FUNCTION_BLOCK FB_Kommunikation
VAR_INPUT
	I_sIP		:STRING;
	SW			:SystemStatusWord;
END_VAR

VAR_OUTPUT
	CW			:SystemControlWord;
	Busy		:BOOL;
	Error		:BOOL;
	ErrorID		:DWORD;
END_VAR

VAR
	Connect				:UA_Connect;
	Disconnect			:UA_Disconnect; 
	Read 				:UA_Read;
	Write				:UA_Write;
	Node				:UA_NodeGetHandle;
	NameSpaceIndex		:UA_GetNamespaceIndex;
	
	ConnectInfo			:ST_UASessionConnectInfo;
	NodeID				:ST_UANodeID;
	NodeInfo			:ST_UANodeAdditionalInfo;
	
	ConnectionHdl		:DWORD;
	NoteHdl				:DWORD;
	NameSpace			:UINT;
	IndexRangeCount		:UINT := 1;
	IndexRange			:ARRAY [1..nMaxIndexRange] OF ST_UAIndexRange;
	NodeIdentifier		:STRING(MAX_STRING_LENGTH) := 'GVL_OPC_UA.SW';
	ReadData			:SystemStatusWord; 		// change to node data type
END_VAR

// Definition der Verbindungsinformationen
ConnectInfo.tSessionTimeout := T#1M;
ConnectInfo.tConnectTimeout := T#1M;
ConnectInfo.sApplicationName := '';
ConnectInfo.eSecurityMode := eUASecurityMsgMode_Sign_Encrypt;				// 3 = Sign_Encrypted
ConnectInfo.eSecurityPolicyUri := eUASecurityPolicy_Basic256Sha256;			// 4 = Basic256  
ConnectInfo.eTransportProfileUri := eUATransportProfileUri_UATcp;			// 1 = UATcp
ConnectInfo.stUserIdentTokenType.eUserIdentTokenType := eUAUITT_Username;	// 1 = Username
ConnectInfo.stUserIdentTokenType.sTokenParam1 := 'Administrator';			// Username
ConnectInfo.stUserIdentTokenType.sTokenParam2 := '1';						// PW

GVL.SW := ReadData;

ACTION ACT_Connect:
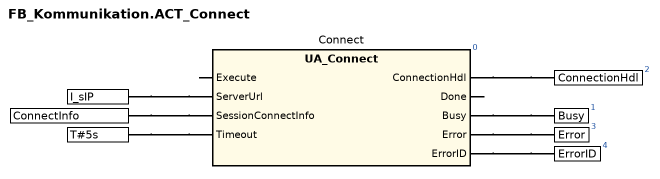
Connect(ServerUrl := I_sIP, SessionConnectInfo := ConnectInfo, Timeout := T#5s); // UA_Connect
Busy := Connect.Busy;
ConnectionHdl := Connect.ConnectionHdl;
Error := Connect.Error;
ErrorID := Connect.ErrorID;
END_ACTION

ACTION ACT_Disconnect:
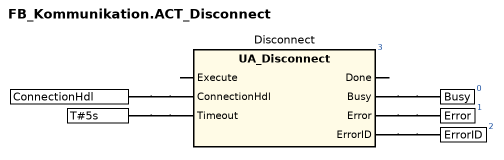
Busy := Disconnect.Busy;
Error := Disconnect.Error;
ErrorID := Disconnect.ErrorID;
Disconnect(ConnectionHdl := ConnectionHdl, Timeout := T#5s); // UA_Disconnect
END_ACTION

ACTION ACT_GetNameSpaceIndex:
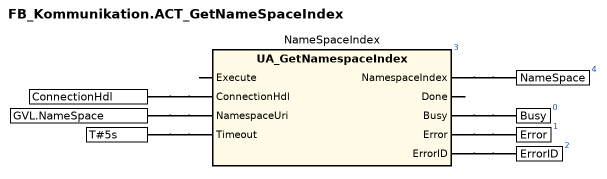
Busy := NameSpaceIndex.Busy;
Error := NameSpaceIndex.Error;
ErrorID := NameSpaceIndex.ErrorID;
NameSpaceIndex(ConnectionHdl := ConnectionHdl, NamespaceUri := GVL.NameSpace, Timeout := T#5s); // UA_GetNamespaceIndex
NameSpace := NameSpaceIndex.NamespaceIndex;
END_ACTION

ACTION ACT_GetNodes:
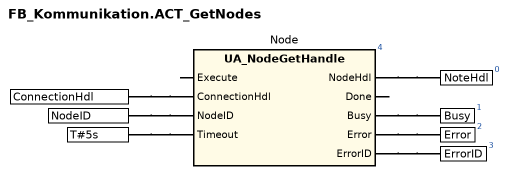
NoteHdl := Node.NodeHdl;
Busy := Node.Busy;
Error := Node.Error;
ErrorID := Node.ErrorID;
Node(ConnectionHdl := ConnectionHdl, NodeID := NodeID, Timeout := T#5s); // UA_NodeGetHandle
END_ACTION

ACTION ACT_Read:
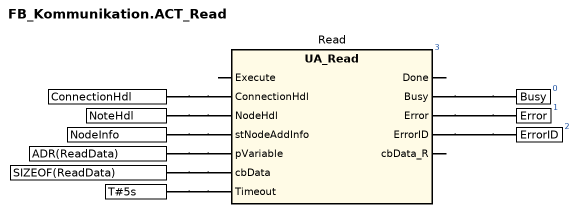
Busy := Read.Busy;
Error := Read.Error;
ErrorID := Read.ErrorID;
Read(
    ConnectionHdl := ConnectionHdl,
    NodeHdl := NoteHdl,
    stNodeAddInfo := NodeInfo,
    pVariable := ADR(ReadData),
    cbData := SIZEOF(ReadData),
    Timeout := T#5s); // UA_Read
END_ACTION

ACTION ACT_Write:
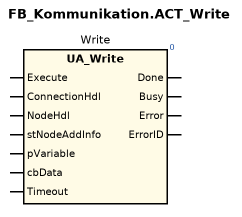
Write(); // UA_Write
END_ACTION

METHOD M_M_Connect : BOOL
VAR_INPUT
END_VAR
// Setzen der Ausführvariabel
Connect.Execute := TRUE;
// Aufrufen der Aktion
ACT_Connect();

// Methode abschliessen
IF Connect.Done THEN
	Connect.Execute := FALSE;
	M_M_Connect := TRUE;
END_IF
END_METHOD

METHOD M_M_Disconnect : BOOL
VAR_INPUT
END_VAR
// Setzen der Ausführvariabel
Disconnect.Execute := TRUE;
// Aufrufen der Aktion
Act_Disconnect();

// Methode abschliessen
IF Disconnect.Done THEN
	Disconnect.Execute := FALSE;
	M_M_Disconnect := TRUE;
END_IF
END_METHOD

METHOD M_M_GetNameSpaceIndex : BOOL
VAR_INPUT
END_VAR
// Setzen der Ausführvariabel
NameSpaceIndex.Execute := TRUE;
// Aufrufen der Aktion
ACT_GetNameSpaceIndex();

// Methode abschliessen
IF NameSpaceIndex.Done THEN
	NameSpaceIndex.Execute := FALSE;
	M_M_GetNameSpaceIndex := TRUE;
END_IF
END_METHOD

METHOD M_M_GetNodes : BOOL
VAR_INPUT
END_VAR
// Definieren von relevanten Parameter
NodeID.eIdentifierType := eUAIdentifierType_String;
NodeID.nNamespaceIndex := NameSpace;
NodeID.sIdentifier := NodeIdentifier;

// Setzen der Ausführvariabel
Node.Execute := TRUE;
// Aufrufen der Aktion
ACT_GetNodes();

// Methode abschliessen
IF Node.Done THEN
	Node.Execute := FALSE;
	M_M_getNodes := TRUE;
END_IF
END_METHOD

METHOD M_M_Read : BOOL
VAR_INPUT
END_VAR
// Definieren von Parametern
//NodeInfo.nIndexRangeCount := IndexRangeCount;
//NodeInfo.stIndexRange := IndexRange;

// Setzen der Ausführvariabel
Read.Execute := TRUE;
// Aufrufen der Aktion
ACT_Read();

// Methode abschliessen
IF Read.Done THEN
	Read.Execute := FALSE;
	M_M_Read := TRUE;
END_IF
END_METHOD

METHOD M_M_Write : BOOL
VAR_INPUT
END_VAR


// Methode abschliessen
IF Write.Done THEN
	Write.Execute := FALSE;
	M_M_Write := TRUE;
END_IF
END_METHOD

END_FUNCTION_BLOCK

(* stored: Version 1.1.0.1, ProductVersion 3.1.4024.12
   POU FB_Kommunikation: Id {f9ca3bd7-2f7d-43be-962a-c929cfd78685}, SpecialFunc None
   Folder 01_Aktionen: Id {fb256ad0-9914-4e4c-8d69-7dd42e1d4202}
   Folder 02_Methoden: Id {4c1c4bc0-f7f9-4deb-bc95-6da45b4305d3}
   Action ACT_Connect: Id {f6a11f60-4fd4-4787-9f03-de252b88edce}
   Action ACT_Disconnect: Id {685bc991-9763-4622-9169-97f6e0e5edc0}
   Action ACT_GetNameSpaceIndex: Id {f8f31d3b-f5e1-4ef4-ad11-6f141c275e19}
   Action ACT_GetNodes: Id {12a20346-972c-43a7-a042-99ea9918371c}
   Action ACT_Read: Id {9f1cfaa9-e461-4a87-9f87-fd7bdfe3f2db}
   Action ACT_Write: Id {a844e75e-a16a-4e6b-9cae-220677a4e810}
   Method M_M_Connect: Id {fbb7e453-0390-494d-834a-96ae116ab685}
   Method M_M_Disconnect: Id {e5b2ce30-0ecf-4aba-a205-34ba1d7de38d}
   Method M_M_GetNameSpaceIndex: Id {65463151-986e-481f-a532-6ad14f7b213a}
   Method M_M_GetNodes: Id {9a44e1af-000b-4d40-b138-9a7a73b00093}
   Method M_M_Read: Id {085aef21-12d2-42ad-bb52-5be058d05602}
   Method M_M_Write: Id {6a10ac80-cbf4-46ff-9454-4b4f3309047a} *)
